SUBAPPLICATION mapping_Uebung_033_VV_FORTE_PC_A (* LED Strip Blinkende LED *)
  (* Standard: 61499-2; Description: Copyright (c) 2023 HR Agrartechnik GmbH This program and the accompanying materials are made available under the terms of the Eclipse Public License 2.0 which is available at https://www.eclipse.org/legal/epl-2.0/ SPDX-License-Identifier: EPL-2.0 *)
  (* Version 1.0, 2023-10-23, Franz Höpfinger, HR Agrartechnik GmbH *)
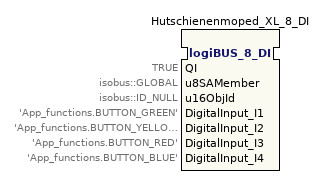
  FBS
    Hutschienenmoped_XL_8_DI : logiBUS_8_DI(QI := TRUE, u8SAMember := isobus::GLOBAL, u16ObjId := isobus::ID_NULL, DigitalInput_I1 := 'App_functions.BUTTON_GREEN', DigitalInput_I2 := 'App_functions.BUTTON_YELLOW', DigitalInput_I3 := 'App_functions.BUTTON_RED', DigitalInput_I4 := 'App_functions.BUTTON_BLUE');
  END_FBS
END_SUBAPPLICATION
